// SIMATIC S7-200 project (STEP 7-Micro/WIN), CPU 221 REL 01.10

ORGANIZATION_BLOCK 主程序:OB1
TITLE=程序注释
BEGIN
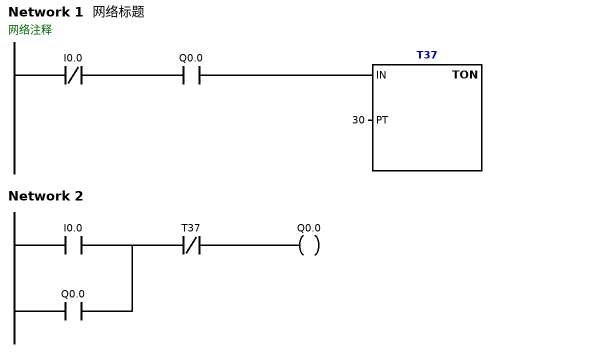
Network 1 // 网络标题
// 网络注释
LDN    I0.0
A      Q0.0
TON    T37, 30
Network 2
LD     I0.0
O      Q0.0
AN     T37
=      Q0.0
END_ORGANIZATION_BLOCK
